FUNCTION_BLOCK FB_Start
VAR_INPUT
END_VAR
VAR_OUTPUT
END_VAR
VAR
	bSwitch AT%I* : BOOL; 
	bLamp   AT%Q* : BOOL; 
nCaseIndex : INT;
	nGleis: BOOL;
END_VAR


bLamp := bSwitch;
CASE nCaseIndex OF 
0: 	
	IF bSwitch = TRUE  THEN
		nCaseIndex := 10; 
	END_IF;; 
	
10: 
	

	IF bSwitch = TRUE  THEN
		nGleis := TRUE;
	
	ELSE
		nGleis := FALSE;
	END_IF;; 
	
END_CASE

END_FUNCTION_BLOCK

(* stored: Version 1.1.0.1
   POU FB_Start: Id {911134b4-3fe5-4ff9-b598-0b0f7a52db32}, SpecialFunc None *)
